# EPICS autosave request: testApp/Db/configMenu.req
$(P)$(CONFIG)Menu:currName
$(P)$(CONFIG)Menu:currDesc
